// TIA Portal project "Reforma Molino FRYMA - Airsa" (V16)

(* hardware
DEVICE "S7-1200 station_1"  S7-1200 Station
   slot 0: "Rack_0"  S7-1200 Rack  Rack  V1.0
   slot 1: "PLC_1"  CPU 1214C DC/DC/DC  6ES7 214-1AG40-0XB0  V4.4
   slot 2: "DI 16x24VDC_1"  6ES7 221-1BH32-0XB0  V2.0
   slot 3: "DQ 16x24VDC_1"  SM 1222 DQ16 x 24VDC  6ES7 222-1BH32-0XB0  V2.0
   slot 4: "AI 4x13BIT/AQ 2x14BIT_1"  6ES7 234-4HE32-0XB0  V2.1
   slot 5: "SIWAREX WP231 Papilla"  SIWAREX WP231  7MH4960-2AA01
   slot 6: "SIWAREX WP231 Aceite"  SIWAREX WP231  7MH4960-2AA01
*)

// ===== PLC "PLC_1"  CPU 1214C DC/DC/DC =====
// protected blocks, not shown: "WP231PR_Aceite", "WP231PR_Papilla"

VAR_GLOBAL   // PLC tag table "Tabla de variables estándar"
   "V1" AT %M0.0 : Bool;   // V Ingreso aceite al tk 5
   "V2" AT %M0.1 : Bool;   // V placa orificio aceite 1kg/s
   "V3" AT %M0.2 : Bool;   // V ingreso aceite desde tk5 hacia molino
   "V4" AT %M0.3 : Bool;   // V ingreso papilla desde tk4 hacia molino
   "V5" AT %M0.4 : Bool;   // V bypass M2
   "V6" AT %M0.5 : Bool;   // V CIP molino
   "V7" AT %M0.6 : Bool;   // V ingreso superior al molino
   "V8" AT %M0.7 : Bool;   // V para recirculación molino
   "V9" AT %M1.0 : Bool;   // V venteo
   "V10" AT %M1.1 : Bool;   // V agua para bomba vacío
   "V11" AT %M1.2 : Bool;   // V antimezcla doble mariposa
   "V12" AT %M1.3 : Bool;   // V desague
   "V13" AT %M1.4 : Bool;   // V recirculación
   "V14" AT %M1.5 : Bool;   // V antimezcla doble mariposa
   "V15" AT %M1.6 : Bool;   // V recirculación
   "V16" AT %M1.7 : Bool;   // V recirculación
   "V17" AT %M2.0 : Bool;   // V recirculación
   "V18" AT %M2.1 : Bool;   // V CIP tk aceite
   "V19" AT %M2.2 : Bool;   // V ingreso agua tk aceite
   "V20" AT %M2.3 : Bool;   // V ingreso papilla tk4
   "V21" AT %M2.4 : Bool;   // V CIP tk papilla
   "Conf_A_V1" AT %M2.5 : Bool;   // Confirmación apertura V1
   "Conf_A_V2" AT %M2.6 : Bool;   // Confirmación apertura V2
   "Conf_A_V3" AT %M2.7 : Bool;   // Confirmación apertura V3
   "Conf_A_V4" AT %M3.0 : Bool;   // Confirmación apertura V4
   "Conf_A_V5" AT %M3.1 : Bool;   // Confirmación apertura V5
   "Conf_A_V6" AT %M3.2 : Bool;   // Confirmación apertura V6
   "Conf_A_V7" AT %M3.3 : Bool;   // Confirmación apertura V7
   "Conf_A_V8" AT %M3.4 : Bool;   // Confirmación apertura V8
   "Conf_A_V9" AT %M3.5 : Bool;   // Confirmación apertura V9
   "Conf_A_V10" AT %M3.6 : Bool;   // Confirmación apertura V10
   "Conf_A_V11" AT %M3.7 : Bool;   // Confirmación apertura V11
   "Conf_A_V12" AT %M4.0 : Bool;   // Confirmación apertura V12
   "Conf_A_V13" AT %M4.1 : Bool;   // Confirmación apertura V13
   "Conf_A_V14" AT %M4.2 : Bool;   // Confirmación apertura V14
   "Conf_A_V15" AT %M4.3 : Bool;   // Confirmación apertura V15
   "Conf_A_V16" AT %M4.4 : Bool;   // Confirmación apertura V16
   "Conf_A_V17" AT %M4.5 : Bool;   // Confirmación apertura V17
   "Conf_A_V18" AT %M4.6 : Bool;   // Confirmación apertura V18
   "Conf_A_V19" AT %M4.7 : Bool;   // Confirmación apertura V19
   "Conf_A_V20" AT %M5.0 : Bool;   // Confirmación apertura V20
   "Conf_A_V21" AT %M5.1 : Bool;   // Confirmación apertura V21
   "Habilita_Gral" AT %M6.0 : Bool;   // Habilitacion general del proceso (HMI)
   "P_Iniciar_Proceso" AT %M6.1 : Bool;   // Pulsador para dar inicio al proceso (HMI)
   "Cond_Arranque_Ok" AT %M6.2 : Bool;   // El sistema no tiene fallas y está listo para comenzar proceso
   "Ciclo_Unico" AT %M6.3 : Bool;   // El sistema producirá un único lote (HMI)
   "Ciclo_Automatico" AT %M6.4 : Bool;   // El sistema producirá lotes de forma continua (HMI)
   "P_Conf_Carga" AT %M6.5 : Bool;   // Pulsador de confirmación de carga de ingredientes (HMI)
   "P_Inicio_Molino" AT %M6.6 : Bool;   // Pulsador para continuar con el transpaso de los tanques hacia el molino (HMI)
   "P_Parada" AT %M6.7 : Bool;   // Pulsador de parada para detener el ciclo de forma inmediata (HMI)
END_VAR

TYPE "UDT_Esc_Analog"
   STRUCT
      Source : Int;
      Input_Min : Int;
      Input_Max : Int;
      Escala_Min : Real;
      Escala_Max : Real;
      Offset : Real;
      Val_Escalado : Real;
      Error : Bool;
   END_STRUCT;
END_TYPE

DATA_BLOCK "Estados del proceso"   // DB2
{ S7_Optimized_Access := 'FALSE' }
VERSION : 0.1
   VAR
      E0 : Bool;   // Estado del diagrama GRAFCET
      E1 : Bool;   // Estado del diagrama GRAFCET
      E2 : Bool;   // Estado del diagrama GRAFCET
      E3 : Bool;   // Estado del diagrama GRAFCET
      E4 : Bool;   // Estado del diagrama GRAFCET
      E5 : Bool;   // Estado del diagrama GRAFCET
      E6 : Bool;   // Estado del diagrama GRAFCET
      E7 : Bool;   // Estado del diagrama GRAFCET
      E8 : Bool;   // Estado del diagrama GRAFCET
      E9 : Bool;   // Estado del diagrama GRAFCET
      E10 : Bool;   // Estado del diagrama GRAFCET
      E11 : Bool;   // Estado del diagrama GRAFCET
      E12 : Bool;   // Estado del diagrama GRAFCET
      E13 : Bool;   // Estado del diagrama GRAFCET
      E14 : Bool;   // Estado del diagrama GRAFCET
   END_VAR
BEGIN
END_DATA_BLOCK

DATA_BLOCK "Set Points proceso actual"   // DB3
{ S7_Optimized_Access := 'FALSE' }
VERSION : 0.1
   VAR
      SP_Peso_Papilla : Real;   // Kg de papilla que se cargarán en el tk4 (HMI)
      SP_Peso_Aceite : Real;   // Kg de aceite que se cargarán en el tk5 (HMI)
      SP_Peso_Ingredientes : Real;   // Kg de ingredientes que se agregarán (HMI)
      SP_Peso_Remanente_Aceite : Real;   // Peso máximo remanente permitido luego del vaciado del tanque de aceite (HMI)
      SP_Peso_Remanente_Papilla : Real;   // Peso máximo remanente permitido luego del vaciado del tanque de papilla (HMI)
      SP_Presion_Vacio_Papilla : Real;   // Sp vacío para carga de papilla (default -600 mBar) (HMI)
      SP_Presion_Vacio_Aceite : Real;   // Sp vacío para carga de aceite (default -700 mBar) (HMI)
      SP_N_Rupturas_Vacio_Papilla : UInt;   // Cantidad de rupturas de vacio al vaciar el tk de papilla(HMI)
      SP_N_Rupturas_Vacio_Aceite : UInt;   // Cantidad de rupturas de vacio al vaciar el tk de aceite(HMI)
   END_VAR
BEGIN
END_DATA_BLOCK

DATA_BLOCK "Recetas"   // DB4
{ S7_Optimized_Access := 'FALSE' }
VERSION : 0.1
BEGIN
END_DATA_BLOCK

DATA_BLOCK "Comandos HMI"   // DB5
{ S7_Optimized_Access := 'FALSE' }
VERSION : 0.1
   VAR
      Habilita_Gral : Bool;   // Habilitacion general del proceso (HMI)
      P_Iniciar_Proceso : Bool;   // Pulsador para dar inicio al proceso (HMI)
      Ciclo_Unico : Bool;   // El sistema producirá un único lote (HMI)
      Ciclo_Automatico : Bool;   // El sistema producirá lotes de forma continua (HMI)
      P_Conf_Carga : Bool;   // Pulsador de confirmación de carga de ingredientes (HMI)
      P_Inicio_Molino : Bool;   // Pulsador para continuar con el transpaso de los tanques hacia el molino (HMI)
      P_Parada : Bool;   // Pulsador de parada para detener el ciclo de forma inmediata (HMI)
      P_Conf_Descarga_Molino : Bool;   // Pulsador para descargar el producto terminado del molino
   END_VAR
BEGIN
END_DATA_BLOCK

DATA_BLOCK "Variables del Proceso"   // DB6
{ S7_Optimized_Access := 'FALSE' }
VERSION : 0.1
   VAR
      Cond_Arranque_Ok : Bool;   // El sistema no tiene fallas y está listo para comenzar proceso
      Tanques_Ok : Bool;   // Los tanques 4 y 5 están vacíos y listos
      Papilla_Lista : Bool;   // La papilla ya está cargada en el tanque y lista para pasar al molino
      Aceite_Listo : Bool;   // El aceite ya está cargado en el tanque junto con sus ingredientes, listo para pasar al molino
      Molino_Listo : Bool;   // El molino se encuentra vacío y listo para procesar un nuevo lote
      Rupturas_Vacio_Actuales : UInt;   // Cantidad de rupturas de vacío al trasladar papilla o aceite al molino
      Estado_Reg_Molino : Bool;   // El molino se encuentra en estado de régimen listo para comenzar la carga de aceite
      Producto_Terminado : Bool;   // El molino terminó de emulsionar y mezclar la mayonesa
   END_VAR
BEGIN
END_DATA_BLOCK

// folder: Analogicas

DATA_BLOCK "Lecturas_Analogicas"   // DB1
{ S7_Optimized_Access := 'FALSE' }
VERSION : 0.1
   VAR
      Balanza_Papilla : Real;
      Balanza_Aceite : Real;
      Temperatura_Molino : "UDT_Esc_Analog";
      Vacuómetro : "UDT_Esc_Analog";
   END_VAR
BEGIN
END_DATA_BLOCK

// folder: E/S Digitales

DATA_BLOCK "Entradas/Salidas Digitales"   // DB7
{ S7_Optimized_Access := 'TRUE' }
VERSION : 0.1
   VAR
      E_Sensor_Nivel_Molino : Bool;
   END_VAR
BEGIN
END_DATA_BLOCK

// folder: System blocks/Program resources

DATA_BLOCK "IEC_Timer_Descarga_DB"   // DB8
{ S7_Optimized_Access := 'TRUE' }
AUTHOR : Simatic
FAMILY : IEC
NAME : IEC_TMR
VERSION : 1.0
// stored: InstanceOfName IEC_TIMER
"IEC_TIMER"
BEGIN
END_DATA_BLOCK

// folder: (top level)

FUNCTION_BLOCK "Lógica del proceso"   // FB1, LAD
{ S7_Optimized_Access := 'TRUE' }
VERSION : 0.1
   VAR_TEMP
      Temp_Carga_Ingredientes : Real;
   END_VAR
BEGIN

REGION Network 1: Set Estado 0:
   // El proceso no está habilitado
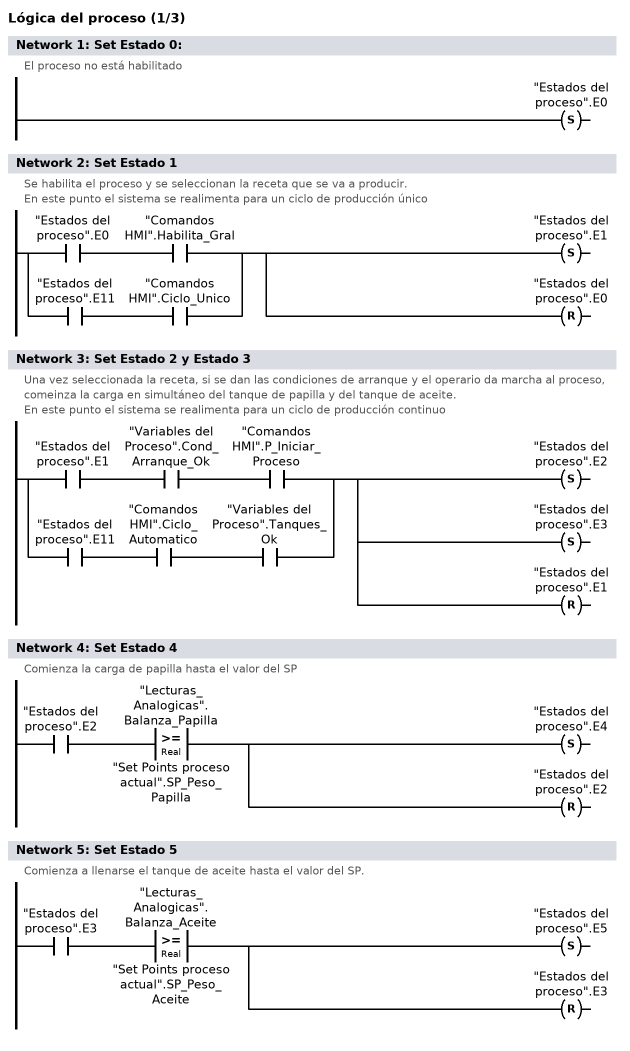
   RUNG wire#powerrail
      S_Coil( "Estados del proceso".E0 )
   END_RUNG
   // the same network as SCL:
   "Estados del proceso".E0 := TRUE;
END_REGION

REGION Network 2: Set Estado 1
   // Se habilita el proceso y se seleccionan la receta que se va a producir.
   // En este punto el sistema se realimenta para un ciclo de producción único
   RUNG wire#powerrail
      Contact( "Estados del proceso".E0 )
      Contact( "Comandos HMI".Habilita_Gral )
      wire#w1
      S_Coil( "Estados del proceso".E1 )
   END_RUNG
   RUNG wire#powerrail
      Contact( "Estados del proceso".E11 )
      Contact( "Comandos HMI".Ciclo_Unico )
   END_RUNG wire#w1
   RUNG wire#w1
      R_Coil( "Estados del proceso".E0 )
   END_RUNG
   // the same network as SCL:
   IF ("Estados del proceso".E0 AND "Comandos HMI".Habilita_Gral) OR ("Estados del proceso".E11 AND "Comandos HMI".Ciclo_Unico) THEN
       "Estados del proceso".E1 := TRUE;
       "Estados del proceso".E0 := FALSE;
   END_IF;
END_REGION

REGION Network 3: Set Estado 2 y Estado 3
   // Una vez seleccionada la receta, si se dan las condiciones de arranque y el operario da marcha al proceso, comeinza la carga en simultáneo del tanque de papilla y del tanque de aceite.
   // En este punto el sistema se realimenta para un ciclo de producción continuo
   RUNG wire#powerrail
      Contact( "Estados del proceso".E1 )
      Contact( "Variables del Proceso".Cond_Arranque_Ok )
      Contact( "Comandos HMI".P_Iniciar_Proceso )
      wire#w1
      S_Coil( "Estados del proceso".E2 )
   END_RUNG
   RUNG wire#powerrail
      Contact( "Estados del proceso".E11 )
      Contact( "Comandos HMI".Ciclo_Automatico )
      Contact( "Variables del Proceso".Tanques_Ok )
   END_RUNG wire#w1
   RUNG wire#w1
      S_Coil( "Estados del proceso".E3 )
   END_RUNG
   RUNG wire#w1
      R_Coil( "Estados del proceso".E1 )
   END_RUNG
   // the same network as SCL:
   IF ("Estados del proceso".E1 AND "Variables del Proceso".Cond_Arranque_Ok AND "Comandos HMI".P_Iniciar_Proceso) OR ("Estados del proceso".E11 AND "Comandos HMI".Ciclo_Automatico AND "Variables del Proceso".Tanques_Ok) THEN
       "Estados del proceso".E2 := TRUE;
       "Estados del proceso".E3 := TRUE;
       "Estados del proceso".E1 := FALSE;
   END_IF;
END_REGION

REGION Network 4: Set Estado 4
   // Comienza la carga de papilla hasta el valor del SP
   RUNG wire#powerrail
      Contact( "Estados del proceso".E2 )
      { S7_Templates := "SrcType := Real" } GE_Contact(in1 := "Lecturas_Analogicas".Balanza_Papilla, in2 := "Set Points proceso actual".SP_Peso_Papilla)
      wire#w1
      S_Coil( "Estados del proceso".E4 )
   END_RUNG
   RUNG wire#w1
      R_Coil( "Estados del proceso".E2 )
   END_RUNG
   // the same network as SCL:
   IF "Estados del proceso".E2 AND ("Lecturas_Analogicas".Balanza_Papilla >= "Set Points proceso actual".SP_Peso_Papilla) THEN
       "Estados del proceso".E4 := TRUE;
       "Estados del proceso".E2 := FALSE;
   END_IF;
END_REGION

REGION Network 5: Set Estado 5
   // Comienza a llenarse el tanque de aceite hasta el valor del SP.
   RUNG wire#powerrail
      Contact( "Estados del proceso".E3 )
      { S7_Templates := "SrcType := Real" } GE_Contact(in1 := "Lecturas_Analogicas".Balanza_Aceite, in2 := "Set Points proceso actual".SP_Peso_Aceite)
      wire#w1
      S_Coil( "Estados del proceso".E5 )
   END_RUNG
   RUNG wire#w1
      R_Coil( "Estados del proceso".E3 )
   END_RUNG
   // the same network as SCL:
   IF "Estados del proceso".E3 AND ("Lecturas_Analogicas".Balanza_Aceite >= "Set Points proceso actual".SP_Peso_Aceite) THEN
       "Estados del proceso".E5 := TRUE;
       "Estados del proceso".E3 := FALSE;
   END_IF;
END_REGION

REGION Network 6: Set Estado 6
   // Se solicita el agregado de ingredientes
   // Se chequea que efectivamente se hayan agregado los ingredientes en el aceite y se espera a la confirmación del operario para continuar
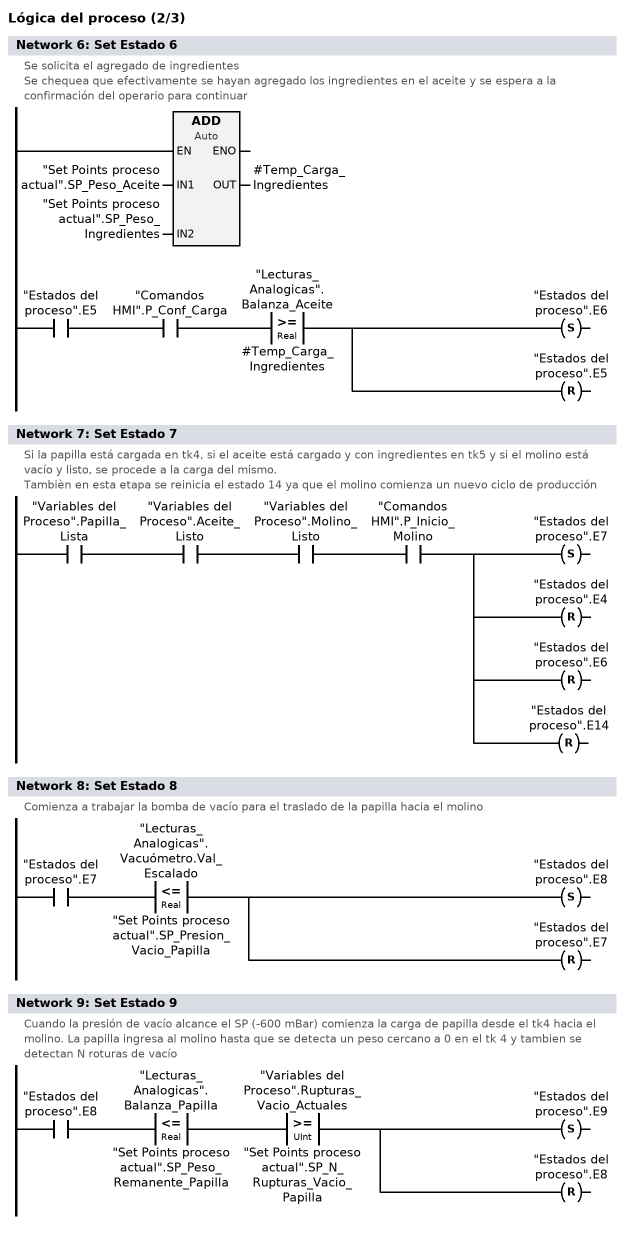
   RUNG wire#powerrail
      Add(in1 := "Set Points proceso actual".SP_Peso_Aceite, in2 := "Set Points proceso actual".SP_Peso_Ingredientes, out => #Temp_Carga_Ingredientes)
   END_RUNG
   RUNG wire#powerrail
      Contact( "Estados del proceso".E5 )
      Contact( "Comandos HMI".P_Conf_Carga )
      { S7_Templates := "SrcType := Real" } GE_Contact(in1 := "Lecturas_Analogicas".Balanza_Aceite, in2 := #Temp_Carga_Ingredientes)
      wire#w1
      S_Coil( "Estados del proceso".E6 )
   END_RUNG
   RUNG wire#w1
      R_Coil( "Estados del proceso".E5 )
   END_RUNG
   // the same network as SCL:
   #Temp_Carga_Ingredientes := "Set Points proceso actual".SP_Peso_Aceite + "Set Points proceso actual".SP_Peso_Ingredientes;
   IF "Estados del proceso".E5 AND "Comandos HMI".P_Conf_Carga AND ("Lecturas_Analogicas".Balanza_Aceite >= #Temp_Carga_Ingredientes) THEN
       "Estados del proceso".E6 := TRUE;
       "Estados del proceso".E5 := FALSE;
   END_IF;
END_REGION

REGION Network 7: Set Estado 7
   // Si la papilla está cargada en tk4, si el aceite está cargado y con ingredientes en tk5 y si el molino está vacío y listo, se procede a la carga del mismo.
   // Tambièn en esta etapa se reinicia el estado 14 ya que el molino comienza un nuevo ciclo de producción
   RUNG wire#powerrail
      Contact( "Variables del Proceso".Papilla_Lista )
      Contact( "Variables del Proceso".Aceite_Listo )
      Contact( "Variables del Proceso".Molino_Listo )
      Contact( "Comandos HMI".P_Inicio_Molino )
      wire#w1
      S_Coil( "Estados del proceso".E7 )
   END_RUNG
   RUNG wire#w1
      R_Coil( "Estados del proceso".E4 )
   END_RUNG
   RUNG wire#w1
      R_Coil( "Estados del proceso".E6 )
   END_RUNG
   RUNG wire#w1
      R_Coil( "Estados del proceso".E14 )
   END_RUNG
   // the same network as SCL:
   IF "Variables del Proceso".Papilla_Lista AND "Variables del Proceso".Aceite_Listo AND "Variables del Proceso".Molino_Listo AND "Comandos HMI".P_Inicio_Molino THEN
       "Estados del proceso".E7 := TRUE;
       "Estados del proceso".E4 := FALSE;
       "Estados del proceso".E6 := FALSE;
       "Estados del proceso".E14 := FALSE;
   END_IF;
END_REGION

REGION Network 8: Set Estado 8
   // Comienza a trabajar la bomba de vacío para el traslado de la papilla hacia el molino
   RUNG wire#powerrail
      Contact( "Estados del proceso".E7 )
      { S7_Templates := "SrcType := Real" } LE_Contact(in1 := "Lecturas_Analogicas".Vacuómetro.Val_Escalado, in2 := "Set Points proceso actual".SP_Presion_Vacio_Papilla)
      wire#w1
      S_Coil( "Estados del proceso".E8 )
   END_RUNG
   RUNG wire#w1
      R_Coil( "Estados del proceso".E7 )
   END_RUNG
   // the same network as SCL:
   IF "Estados del proceso".E7 AND ("Lecturas_Analogicas".Vacuómetro.Val_Escalado <= "Set Points proceso actual".SP_Presion_Vacio_Papilla) THEN
       "Estados del proceso".E8 := TRUE;
       "Estados del proceso".E7 := FALSE;
   END_IF;
END_REGION

REGION Network 9: Set Estado 9
   // Cuando la presión de vacío alcance el SP (-600 mBar) comienza la carga de papilla desde el tk4 hacia el molino. La papilla ingresa al molino hasta que se detecta un peso cercano a 0 en el tk 4 y tambien se detectan N roturas de vacío
   RUNG wire#powerrail
      Contact( "Estados del proceso".E8 )
      { S7_Templates := "SrcType := Real" } LE_Contact(in1 := "Lecturas_Analogicas".Balanza_Papilla, in2 := "Set Points proceso actual".SP_Peso_Remanente_Papilla)
      { S7_Templates := "SrcType := UInt" } GE_Contact(in1 := "Variables del Proceso".Rupturas_Vacio_Actuales, in2 := "Set Points proceso actual".SP_N_Rupturas_Vacio_Papilla)
      wire#w1
      S_Coil( "Estados del proceso".E9 )
   END_RUNG
   RUNG wire#w1
      R_Coil( "Estados del proceso".E8 )
   END_RUNG
   // the same network as SCL:
   IF "Estados del proceso".E8 AND ("Lecturas_Analogicas".Balanza_Papilla <= "Set Points proceso actual".SP_Peso_Remanente_Papilla) AND ("Variables del Proceso".Rupturas_Vacio_Actuales >= "Set Points proceso actual".SP_N_Rupturas_Vacio_Papilla) THEN
       "Estados del proceso".E9 := TRUE;
       "Estados del proceso".E8 := FALSE;
   END_IF;
END_REGION

REGION Network 10: Set Estado 10
   // Una vez cargada la papilla, se la recircula durante un tiempo con el emulsionador encendido hasta llegar  a un estado de régimen. A su vez, se requiere una presion de vacío determinada por el SP  (-700 mBar) para el ingreso de aceite
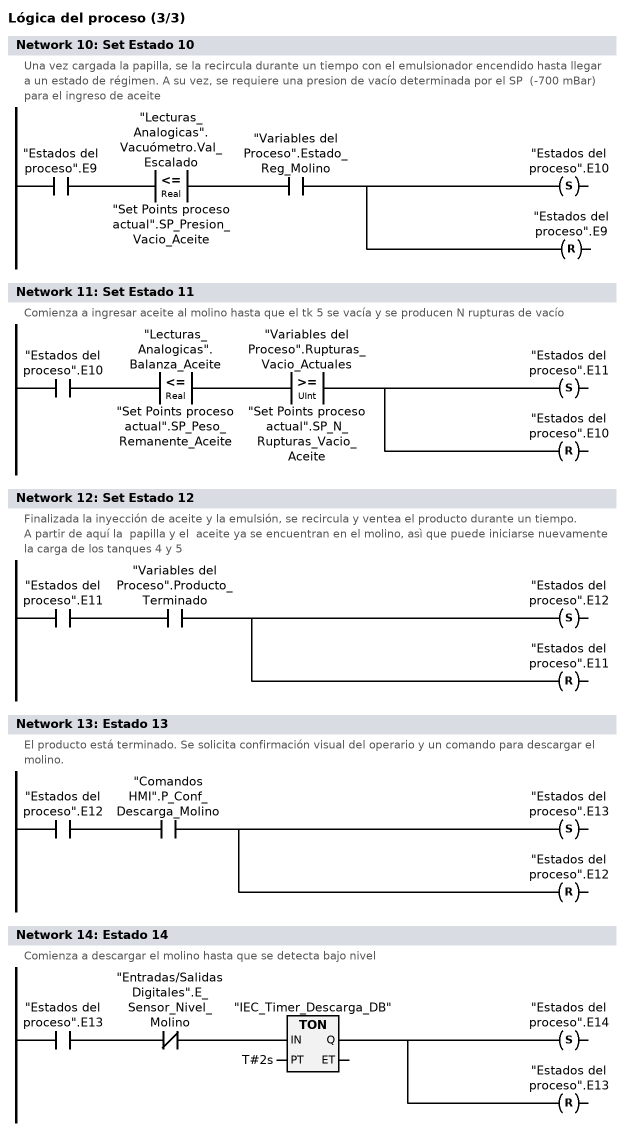
   RUNG wire#powerrail
      Contact( "Estados del proceso".E9 )
      { S7_Templates := "SrcType := Real" } LE_Contact(in1 := "Lecturas_Analogicas".Vacuómetro.Val_Escalado, in2 := "Set Points proceso actual".SP_Presion_Vacio_Aceite)
      Contact( "Variables del Proceso".Estado_Reg_Molino )
      wire#w1
      S_Coil( "Estados del proceso".E10 )
   END_RUNG
   RUNG wire#w1
      R_Coil( "Estados del proceso".E9 )
   END_RUNG
   // the same network as SCL:
   IF "Estados del proceso".E9 AND ("Lecturas_Analogicas".Vacuómetro.Val_Escalado <= "Set Points proceso actual".SP_Presion_Vacio_Aceite) AND "Variables del Proceso".Estado_Reg_Molino THEN
       "Estados del proceso".E10 := TRUE;
       "Estados del proceso".E9 := FALSE;
   END_IF;
END_REGION

REGION Network 11: Set Estado 11
   // Comienza a ingresar aceite al molino hasta que el tk 5 se vacía y se producen N rupturas de vacío
   RUNG wire#powerrail
      Contact( "Estados del proceso".E10 )
      { S7_Templates := "SrcType := Real" } LE_Contact(in1 := "Lecturas_Analogicas".Balanza_Aceite, in2 := "Set Points proceso actual".SP_Peso_Remanente_Aceite)
      { S7_Templates := "SrcType := UInt" } GE_Contact(in1 := "Variables del Proceso".Rupturas_Vacio_Actuales, in2 := "Set Points proceso actual".SP_N_Rupturas_Vacio_Aceite)
      wire#w1
      S_Coil( "Estados del proceso".E11 )
   END_RUNG
   RUNG wire#w1
      R_Coil( "Estados del proceso".E10 )
   END_RUNG
   // the same network as SCL:
   IF "Estados del proceso".E10 AND ("Lecturas_Analogicas".Balanza_Aceite <= "Set Points proceso actual".SP_Peso_Remanente_Aceite) AND ("Variables del Proceso".Rupturas_Vacio_Actuales >= "Set Points proceso actual".SP_N_Rupturas_Vacio_Aceite) THEN
       "Estados del proceso".E11 := TRUE;
       "Estados del proceso".E10 := FALSE;
   END_IF;
END_REGION

REGION Network 12: Set Estado 12
   // Finalizada la inyección de aceite y la emulsión, se recircula y ventea el producto durante un tiempo.
   // A partir de aquí la  papilla y el  aceite ya se encuentran en el molino, asì que puede iniciarse nuevamente la carga de los tanques 4 y 5
   RUNG wire#powerrail
      Contact( "Estados del proceso".E11 )
      Contact( "Variables del Proceso".Producto_Terminado )
      wire#w1
      S_Coil( "Estados del proceso".E12 )
   END_RUNG
   RUNG wire#w1
      R_Coil( "Estados del proceso".E11 )
   END_RUNG
   // the same network as SCL:
   IF "Estados del proceso".E11 AND "Variables del Proceso".Producto_Terminado THEN
       "Estados del proceso".E12 := TRUE;
       "Estados del proceso".E11 := FALSE;
   END_IF;
END_REGION

REGION Network 13: Estado 13
   // El producto está terminado. Se solicita confirmación visual del operario y un comando para descargar el molino.
   RUNG wire#powerrail
      Contact( "Estados del proceso".E12 )
      Contact( "Comandos HMI".P_Conf_Descarga_Molino )
      wire#w1
      S_Coil( "Estados del proceso".E13 )
   END_RUNG
   RUNG wire#w1
      R_Coil( "Estados del proceso".E12 )
   END_RUNG
   // the same network as SCL:
   IF "Estados del proceso".E12 AND "Comandos HMI".P_Conf_Descarga_Molino THEN
       "Estados del proceso".E13 := TRUE;
       "Estados del proceso".E12 := FALSE;
   END_IF;
END_REGION

REGION Network 14: Estado 14
   // Comienza a descargar el molino hasta que se detecta bajo nivel
   "IEC_Timer_Descarga_DB".TON(IN := "Estados del proceso".E13 AND NOT "Entradas/Salidas Digitales".E_Sensor_Nivel_Molino,
                           PT := T#2s);
   IF "IEC_Timer_Descarga_DB".Q THEN
       "Estados del proceso".E14 := TRUE;
       "Estados del proceso".E13 := FALSE;
   END_IF;
END_REGION

REGION Network 15: Fin de ciclo
END_REGION
END_FUNCTION_BLOCK

ORGANIZATION_BLOCK "Main"   // OB1, LAD, ProgramCycle
TITLE = "Main Program Sweep (Cycle)"
{ S7_Optimized_Access := 'TRUE' }
VERSION : 0.1
   VAR_INPUT
      Initial_Call : Bool;   // Initial call of this OB
      Remanence : Bool;   // =True, if remanent data are available
   END_VAR
   VAR_TEMP
      "Lifebit Papilla" : Bool;
      "Lifebit Aceite" : Bool;
   END_VAR
BEGIN

REGION Network 1: Lecturas y conversiones analógicas
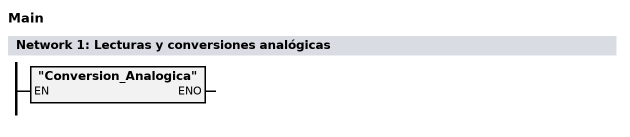
   RUNG wire#powerrail
      "Conversion_Analogica"()
   END_RUNG
   // the same network as SCL:
   "Conversion_Analogica"();
END_REGION
END_ORGANIZATION_BLOCK

// folder: Analogicas

FUNCTION "Macro_Analogico" : Void   // FC1, LAD
{ S7_Optimized_Access := 'TRUE' }
VERSION : 0.1
   VAR_INPUT
      Source : Int;
      Input_Min : Int;
      Input_Max : Int;
      Esc_Min : Real;
      Esc_max : Real;
      Offset : Real;
   END_VAR
   VAR_OUTPUT
      Val_Esc : Real;
      Error : Bool;
   END_VAR
   VAR_TEMP
      Temp0 : Real;
      Temp1 : Real;
   END_VAR
BEGIN

REGION Network 1
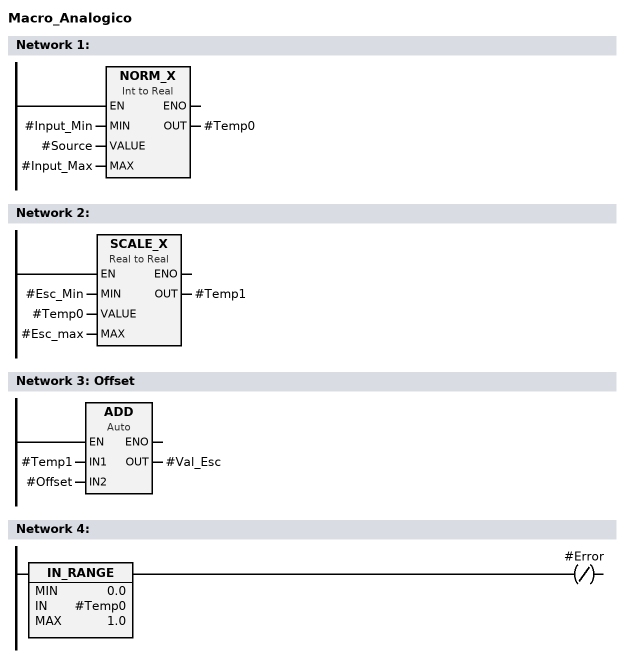
   RUNG wire#powerrail
      { S7_Templates := "[SrcType := Int, DestType := Real]" } Normalize(min := #Input_Min, value := #Source, max := #Input_Max, out => #Temp0)
   END_RUNG
   // the same network as SCL:
   #Temp0 := NORM_X(MIN := #Input_Min, VALUE := #Source, MAX := #Input_Max);
END_REGION

REGION Network 2
   RUNG wire#powerrail
      { S7_Templates := "[SrcType := Real, DestType := Real]" } Scale(min := #Esc_Min, value := #Temp0, max := #Esc_max, out => #Temp1)
   END_RUNG
   // the same network as SCL:
   #Temp1 := SCALE_X(MIN := #Esc_Min, VALUE := #Temp0, MAX := #Esc_max);
END_REGION

REGION Network 3: Offset
   RUNG wire#powerrail
      Add(in1 := #Temp1, in2 := #Offset, out => #Val_Esc)
   END_RUNG
   // the same network as SCL:
   #Val_Esc := #Temp1 + #Offset;
END_REGION

REGION Network 4
   RUNG wire#powerrail
      { S7_Templates := "SrcType := Real" } InRange(min := 0.0, in := #Temp0, max := 1.0)
      I_Coil( #Error )
   END_RUNG
   // the same network as SCL:
   #Error := NOT ((0.0 <= #Temp0) AND (#Temp0 <= 1.0));
END_REGION
END_FUNCTION

FUNCTION "Conversion_Analogica" : Void   // FC2, LAD
TITLE = LECTURAS ANALÓGICAS
{ S7_Optimized_Access := 'TRUE' }
VERSION : 0.1
// Aquí se tratan todas las lecturas analógicas y se obtiene la variable que se utilizará en el programa
   VAR_TEMP
      "Lifebit Papilla" : Bool;
      "Lifebit Aceite" : Bool;
   END_VAR
BEGIN

REGION Network 1: Balanza papilla
   // Este bloque se obtuvo de un archivo de librerias de siemens. Se le asigna la direccion del modulo siwarex declarado en hardware
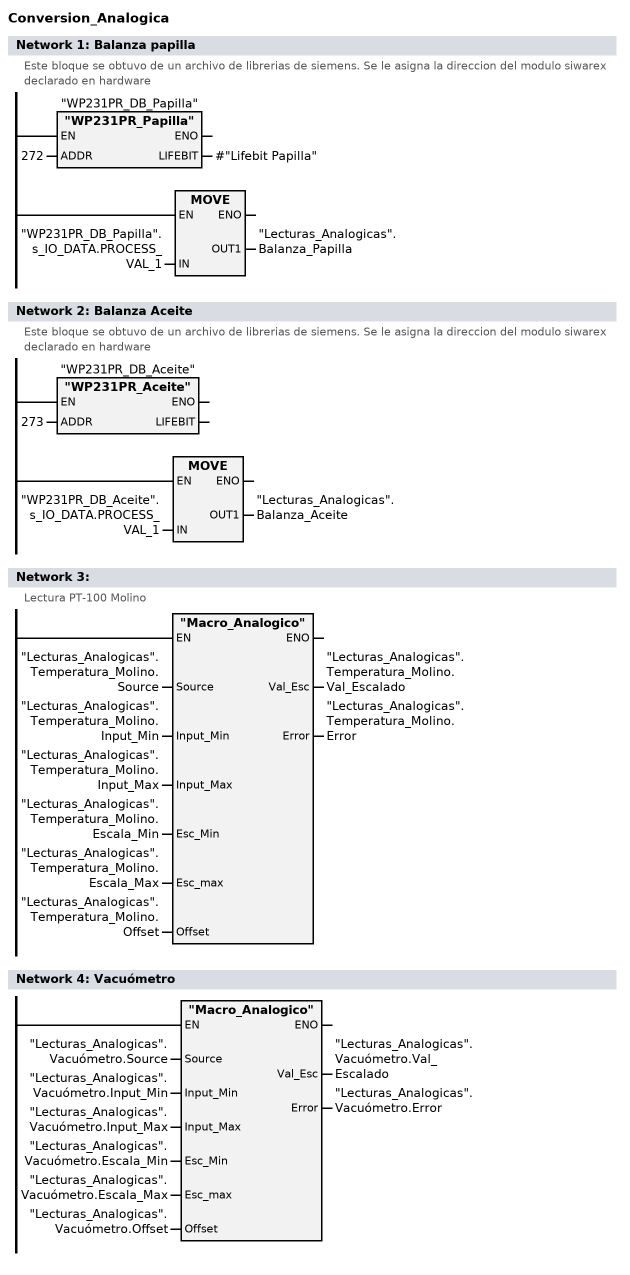
   RUNG wire#powerrail
      "WP231PR_DB_Papilla"(ADDR := 272, LIFEBIT => #"Lifebit Papilla")
   END_RUNG
   RUNG wire#powerrail
      Move(in := "WP231PR_DB_Papilla".s_IO_DATA.PROCESS_VAL_1, out1 => "Lecturas_Analogicas".Balanza_Papilla)
   END_RUNG
   // the same network as SCL:
   "WP231PR_DB_Papilla"(ADDR := 272, LIFEBIT => #"Lifebit Papilla");   // "WP231PR_Papilla"
   "Lecturas_Analogicas".Balanza_Papilla := "WP231PR_DB_Papilla".s_IO_DATA.PROCESS_VAL_1;
END_REGION

REGION Network 2: Balanza Aceite
   // Este bloque se obtuvo de un archivo de librerias de siemens. Se le asigna la direccion del modulo siwarex declarado en hardware
   RUNG wire#powerrail
      "WP231PR_DB_Aceite"(ADDR := 273, LIFEBIT =>)
   END_RUNG
   RUNG wire#powerrail
      Move(in := "WP231PR_DB_Aceite".s_IO_DATA.PROCESS_VAL_1, out1 => "Lecturas_Analogicas".Balanza_Aceite)
   END_RUNG
   // the same network as SCL:
   "WP231PR_DB_Aceite"(ADDR := 273);   // "WP231PR_Aceite"
   "Lecturas_Analogicas".Balanza_Aceite := "WP231PR_DB_Aceite".s_IO_DATA.PROCESS_VAL_1;
END_REGION

REGION Network 3
   // Lectura PT-100 Molino
   RUNG wire#powerrail
      "Macro_Analogico"(Source := "Lecturas_Analogicas".Temperatura_Molino.Source, Input_Min := "Lecturas_Analogicas".Temperatura_Molino.Input_Min, Input_Max := "Lecturas_Analogicas".Temperatura_Molino.Input_Max, Esc_Min := "Lecturas_Analogicas".Temperatura_Molino.Escala_Min, Esc_max := "Lecturas_Analogicas".Temperatura_Molino.Escala_Max, Offset := "Lecturas_Analogicas".Temperatura_Molino.Offset, Val_Esc => "Lecturas_Analogicas".Temperatura_Molino.Val_Escalado, Error => "Lecturas_Analogicas".Temperatura_Molino.Error)
   END_RUNG
   // the same network as SCL:
   "Macro_Analogico"(Source := "Lecturas_Analogicas".Temperatura_Molino.Source,
                     Input_Min := "Lecturas_Analogicas".Temperatura_Molino.Input_Min,
                     Input_Max := "Lecturas_Analogicas".Temperatura_Molino.Input_Max,
                     Esc_Min := "Lecturas_Analogicas".Temperatura_Molino.Escala_Min,
                     Esc_max := "Lecturas_Analogicas".Temperatura_Molino.Escala_Max,
                     Offset := "Lecturas_Analogicas".Temperatura_Molino.Offset,
                     Val_Esc => "Lecturas_Analogicas".Temperatura_Molino.Val_Escalado,
                     Error => "Lecturas_Analogicas".Temperatura_Molino.Error);
END_REGION

REGION Network 4: Vacuómetro
   RUNG wire#powerrail
      "Macro_Analogico"(Source := "Lecturas_Analogicas".Vacuómetro.Source, Input_Min := "Lecturas_Analogicas".Vacuómetro.Input_Min, Input_Max := "Lecturas_Analogicas".Vacuómetro.Input_Max, Esc_Min := "Lecturas_Analogicas".Vacuómetro.Escala_Min, Esc_max := "Lecturas_Analogicas".Vacuómetro.Escala_Max, Offset := "Lecturas_Analogicas".Vacuómetro.Offset, Val_Esc => "Lecturas_Analogicas".Vacuómetro.Val_Escalado, Error => "Lecturas_Analogicas".Vacuómetro.Error)
   END_RUNG
   // the same network as SCL:
   "Macro_Analogico"(Source := "Lecturas_Analogicas".Vacuómetro.Source,
                     Input_Min := "Lecturas_Analogicas".Vacuómetro.Input_Min,
                     Input_Max := "Lecturas_Analogicas".Vacuómetro.Input_Max,
                     Esc_Min := "Lecturas_Analogicas".Vacuómetro.Escala_Min,
                     Esc_max := "Lecturas_Analogicas".Vacuómetro.Escala_Max,
                     Offset := "Lecturas_Analogicas".Vacuómetro.Offset,
                     Val_Esc => "Lecturas_Analogicas".Vacuómetro.Val_Escalado,
                     Error => "Lecturas_Analogicas".Vacuómetro.Error);
END_REGION
END_FUNCTION

// folder: Subprocesos

FUNCTION_BLOCK "Rupturas de vacío"   // FB2, LAD
{ S7_Optimized_Access := 'TRUE' }
VERSION : 0.1
BEGIN
END_FUNCTION_BLOCK